FUNCTION_BLOCK CONVEYOR_WITH_COUNTER (* Extracted Composite Function Block Type *)
  (* Standard: 61499-2 *)
  (* Version 1/9/2023, brink *)
  PACKAGE UAO.Hackathon;
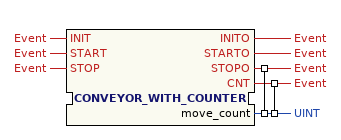
  EVENT_INPUT
    INIT; (* Initialization request *)
    START; (* Start motor & reset counter *)
    STOP; (* Stop motor *)
  END_EVENT
  EVENT_OUTPUT
    INITO; (* Initialization response *)
    STARTO; (* Motor started *)
    STOPO WITH move_count; (* Motor stopped *)
    CNT WITH move_count; (* Count pulse. Fired on every raising AND falling edge of the sensor signal. *)
  END_EVENT
  VAR_OUTPUT
    move_count : UINT; (* Number of pulses(edges) that conveyor moved since last START *)
  END_VAR
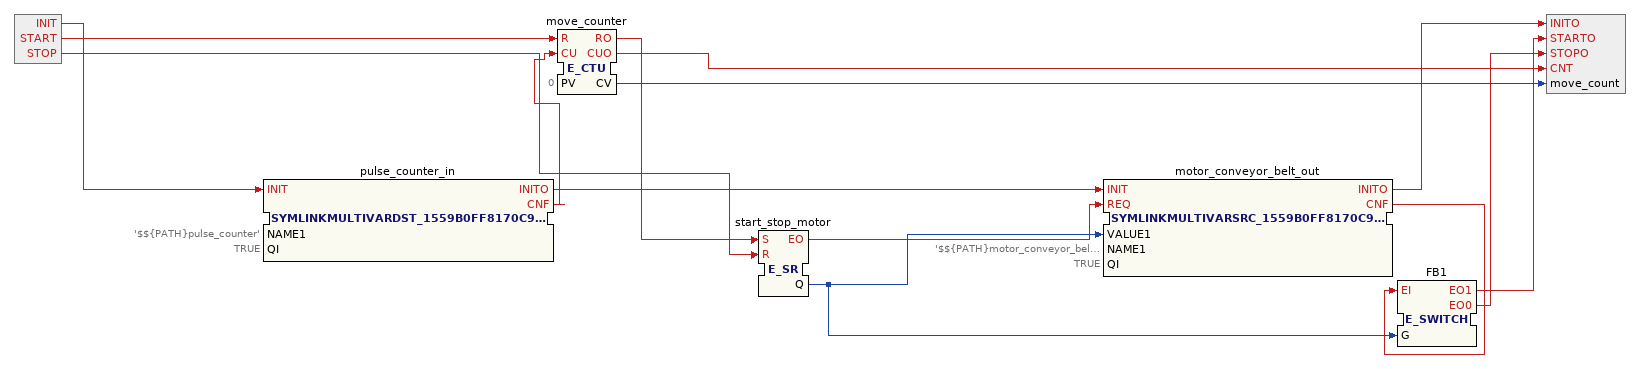
  FBS
    pulse_counter_in : SYMLINKMULTIVARDST_1559B0FF8170C9BA0(NAME1 := '$${PATH}pulse_counter', QI := TRUE); {SET_ATTRIBUTE(Configuration.GenericFBType.InterfaceParams, Runtime.System#I:=1;VALUE${I$}:BOOL)}
    motor_conveyor_belt_out : SYMLINKMULTIVARSRC_1559B0FF8170C9BA0(NAME1 := '$${PATH}motor_conveyor_belt', QI := TRUE); {SET_ATTRIBUTE(Configuration.GenericFBType.InterfaceParams, Runtime.System#I:=1;VALUE${I$}:BOOL)}
    move_counter : E_CTU(PV := 0);
    start_stop_motor : E_SR;
    FB1 : E_SWITCH;
  END_FBS
  EVENT_CONNECTIONS
    pulse_counter_in.INITO TO motor_conveyor_belt_out.INIT;
    INIT TO pulse_counter_in.INIT;
    motor_conveyor_belt_out.INITO TO INITO;
    start_stop_motor.EO TO motor_conveyor_belt_out.REQ;
    START TO move_counter.R;
    motor_conveyor_belt_out.CNF TO FB1.EI;
    FB1.EO1 TO STARTO;
    FB1.EO0 TO STOPO;
    move_counter.RO TO start_stop_motor.S;
    STOP TO start_stop_motor.R;
    pulse_counter_in.CNF TO move_counter.CU;
    move_counter.CUO TO CNT;
  END_CONNECTIONS
  DATA_CONNECTIONS
    start_stop_motor.Q TO motor_conveyor_belt_out.VALUE1;
    move_counter.CV TO move_count;
    start_stop_motor.Q TO FB1.G;
  END_CONNECTIONS
END_FUNCTION_BLOCK
